TYPE Erreur_StructVisu :
STRUCT
	TypeDefaut : STRING(3);
	IDMessage : INT;
	DateMessage : STRING(200);
END_STRUCT
END_TYPE

(* stored: Version 1.1.0.1, ProductVersion 3.1.4024.15
   DUT Erreur_StructVisu: Id {e0741b2f-db12-4026-bddf-07e74233d319} *)
